// TIA Portal V18 export
VAR_GLOBAL   // PLC tag table "Tag table_1"
   nnn1 AT %MD10 : DInt;
   nnn2 AT %MD14 : DInt;
   nnn3 AT %MD18 : DInt;
   nnn4 AT %MD22 : DInt;
   nnn5 AT %MD26 : DInt;
   nnn6 AT %MD30 : DInt;
   nnn7 AT %MD34 : DInt;
   nnn8 AT %MD38 : DInt;
   nnn9 AT %MD42 : DInt;
END_VAR
